(* Logix 5000 project; controller ChiaDynamix_PLC2 Emulate 5570 rev 30.12; software revision 30.00 *)

TASK T00_MainTask (continuous, watchdog 500 ms) : P00_MainProgram

MODULES
   Local : Emulate 5570 (ICP 5, rev 30.12)
      Entradas_Digitales : 1756-IB16 (ICP 3, rev 3.1, Input RPI 20 ms)
      Salidas_Digitales : vendor 1 type 7 code 16 (ICP 4, rev 3.1, Output RPI 20 ms)
      ChiaDynamix_PLC1 : Emulate 5570 (ICP 2, rev 30.1, $a5fb9b3a$ RPI 20 ms, $af09fea8$ RPI 20 ms)
      PLC_Seguridad : Emulate 5570 (ICP 6, rev 30.1, $68d98553$ RPI 20 ms)
END_MODULES

VAR_GLOBAL   (* controller tags *)
   Controles_Permisivos_Consumido : DINT;   // Señal de Seguridad que se recibe del PLC Seguridad
   COUNT : COUNTER[6] := ([0].PRE := 3, [0].ACC := 2, [1].PRE := 3, [1].ACC := 2);
        [1]   // Contador de Cajas Apiladas
        [0]   // Contador de Baldosas Apiladas
   Count_Baldosas_Producido : DINT; {produced}   // Señal que indica que el contador de baldosas ha sido alcanzado
   Count_Cajas_Producido : DINT; {produced}   // Señal que indica cuando el contador de cajas ha sido alcanzado
   FAB_CER_EME_002 : DINT; {produced}   // Botón de Emergencia del PLC2
   FAB_CER_HOMBRE_MUERTO_Producido : DINT; {produced}   // Dead Man Switch
   FAB_CER_RES_002 : DINT; {produced}   // Botón de Reset del PLC2
   FAB_CER_SCANNER_AREA_Producido : DINT; {produced}   // Scanner Area
   FAB_CER_STP_002 : DINT; {produced}   // Botón de Parada del PLC2
   FAB_CER_STR_002 : ALIAS FOR Local:3:I.Data.3;   // Botón de Start del PLC2
   FAB_CORTINAS_SEGURIDAD2_Producido : DINT; {produced}   // Cortinas de seguridad del PLC2
   FAB_INTERLOCK_PUERTA1_Producido : DINT; {produced}   // Interlock Puerta 1
   FAB_INTERLOCK_PUERTA2_Producido : DINT; {produced}   // Interlock Puerta 2
   MA_APILADO1 : ALIAS FOR Local:4:I.Data.6;   // Máquina Apiladora
   MA_EMPA : ALIAS FOR Local:4:I.Data.5;   // Máquina empacadora
   MA_QUAL : ALIAS FOR Local:4:I.Data.4;   // Máquina Qualitron
   MA_VINIPEL : ALIAS FOR Local:4:I.Data.3;   // Máquina Vinipel
   MOT_BAND_001 : ALIAS FOR Local:4:I.Data.2;   // Motor Banda transportadora
   MOT_BAND_DEF : ALIAS FOR Local:4:I.Data.1;   // Motor de banda transportadora de defectos
   MOT_BIFUR : ALIAS FOR Local:4:I.Data.0;   // Motor Palanca de Bifurcación
   POS_BAN_ROBOT2 : ALIAS FOR Local:3:I.Data.13;   // Sensor de posición ubicado en Robot
   POS_BAND_APILADOR : ALIAS FOR Local:3:I.Data.7;   // Sensor de posición ubicado en banda de la máquina apiladora
   POS_BAND_CAJA : ALIAS FOR Local:3:I.Data.6;   // Sensor de posición ubicado en banda del empacado de cajas
   POS_BAND_DEF : ALIAS FOR Local:3:I.Data.5;   // Sensor de posición ubicado en final de banda de defectuosos
   POS_BAND_QUAL : ALIAS FOR Local:3:I.Data.4;   // Sensor de posición ubicado en banda del proceso de Qualitron
   Q : BOOL[32] := ([10] := 1);
        [11]   // Memorias Virtual que activa Motor
        [14]   // Memorias Virtual que activa Motor
        [12]   // Memoria Virtual que activa palanca de bifurcación
        [15]   // Memoria Virtual que activa Máquina Empacadora
   Q10_Producido : DINT; {produced}   // Memoria virtual que activa Máquina Qualitrón
   Q13_Producido : DINT; {produced}   // Memoria Virtual activa Máquina Apiladora
   Q155 : BOOL;   // Memorias Virtual que activa Motor
   Q16_Producido : DINT; {produced}   // Memoria Virtual que activa Rutina del Robot
   Q17_Producido : DINT; {produced}   // Memoria virtual que activa máquina de Vinipel
   Q1_Consumido : DINT;   // Memoria Virtual Q1 que se recibe del PLC1
   Q9_Consumido : DINT;   // Memoria Virtual Q9 que se consume del PLC1
   ROUT_ROBOT2 : ALIAS FOR Local:4:I.Data.7;   // Rutina de Robot 2
   SIGNAL_APILADO1 : DINT; {produced}   // Señal que indica que rutina del Robot 1 ha sido finalizada
   SIGNAL_DEFECT : INT;   // 1: Baldosa NO tiene defecto 2: Baldosa SI tiene defecto
   SIGNAL_ECOPLAT : DINT; {produced}   // Señal que indica que el proceso de máquina de Vinipel ha finalizado
   SIGNAL_EMPA : BOOL;   // Señal que indica que el proceso de empacado finalizó
   SIGNAL_ROUT2 : DINT; {produced}   // Señal que indica que rutina del Robot 2 ha sido finalizada
   SIGNAL_STP : BOOL;   // Señal que indica que el botón de paro está activo
   TIMER : TIMER[6] := ([0].PRE := 30000, [1].PRE := 30000);
        [0]   // Timer de Proceso de Impresión
        [1]   // Timer de Proceso de Secado (Horno)
END_VAR

PROGRAM P00_MainProgram   (* main routine R00_MainRoutine *)

ROUTINE R00_MainRoutine   (* ladder *)
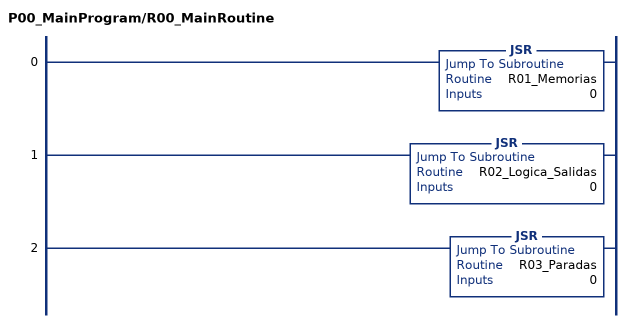
   0: JSR(R01_Memorias,0);
   1: JSR(R02_Logica_Salidas,0);
   2: JSR(R03_Paradas,0);
END_ROUTINE

ROUTINE R01_Memorias   (* ladder *)
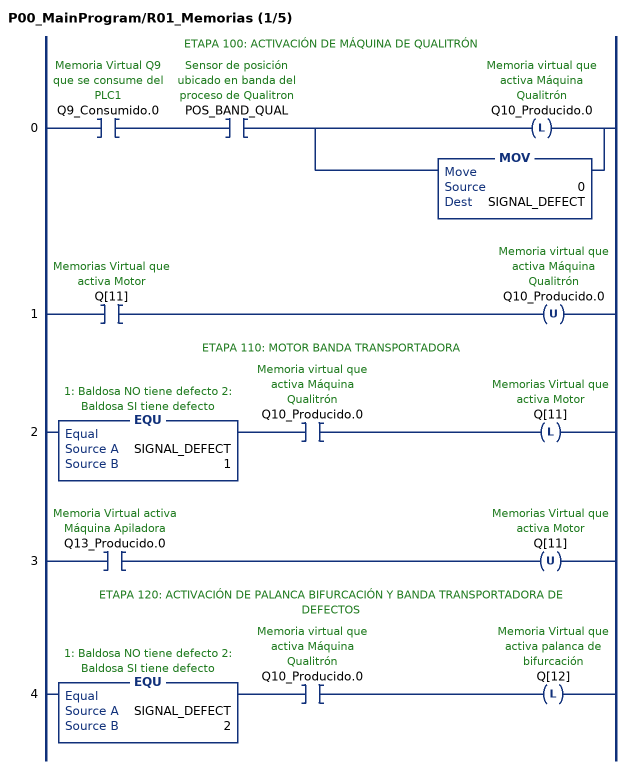
   // ETAPA 100: ACTIVACIÓN DE MÁQUINA DE QUALITRÓN
   0: XIC(Q9_Consumido.0)XIC(POS_BAND_QUAL)[OTL(Q10_Producido.0) ,MOV(0,SIGNAL_DEFECT) ];
   1: XIC(Q[11])OTU(Q10_Producido.0);
   // ETAPA 110: MOTOR BANDA TRANSPORTADORA
   2: EQU(SIGNAL_DEFECT,1)XIC(Q10_Producido.0)OTL(Q[11]);
   3: XIC(Q13_Producido.0)OTU(Q[11]);
   // ETAPA 120: ACTIVACIÓN DE PALANCA BIFURCACIÓN Y BANDA TRANSPORTADORA DE DEFECTOS
   4: EQU(SIGNAL_DEFECT,2)XIC(Q10_Producido.0)OTL(Q[12]);
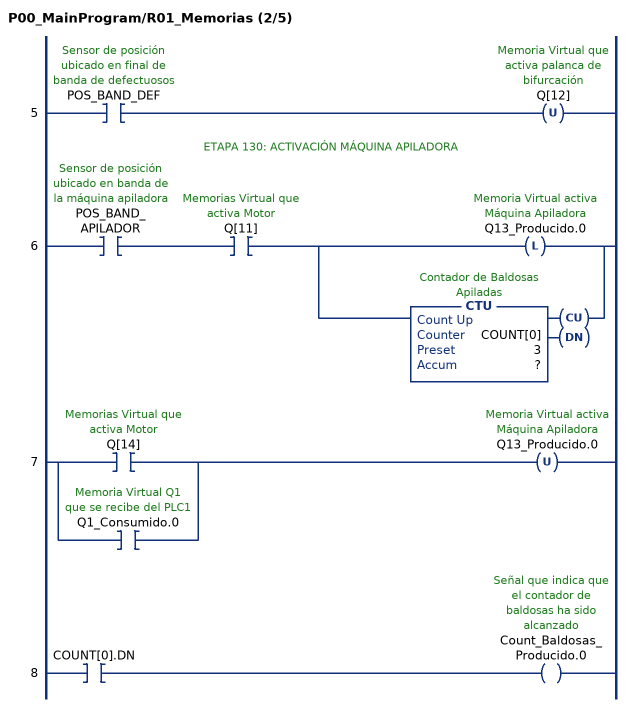
   5: XIC(POS_BAND_DEF)OTU(Q[12]);
   // ETAPA 130: ACTIVACIÓN MÁQUINA APILADORA
   6: XIC(POS_BAND_APILADOR)XIC(Q[11])[OTL(Q13_Producido.0) ,CTU(COUNT[0],?,?) ];
   7: [XIC(Q[14]) ,XIC(Q1_Consumido.0) ]OTU(Q13_Producido.0);
   8: XIC(COUNT[0].DN)OTE(Count_Baldosas_Producido.0);
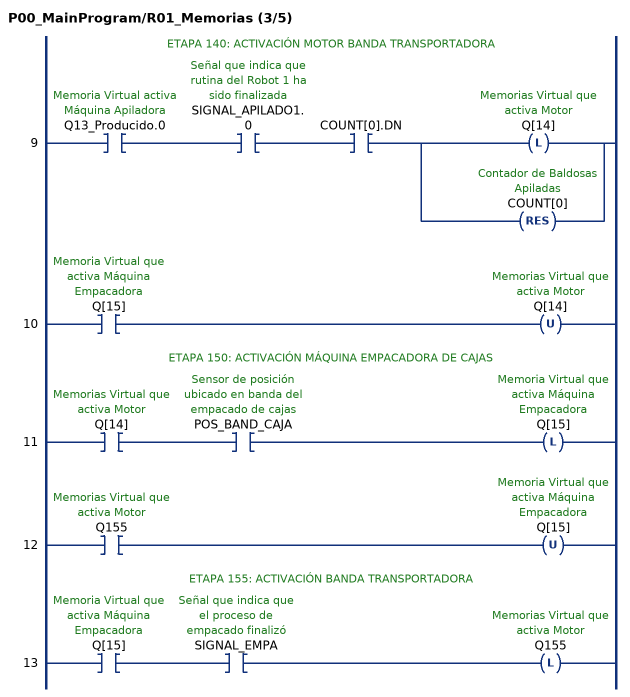
   // ETAPA 140: ACTIVACIÓN MOTOR BANDA TRANSPORTADORA
   9: XIC(Q13_Producido.0)XIC(SIGNAL_APILADO1.0)XIC(COUNT[0].DN)[OTL(Q[14]) ,RES(COUNT[0]) ];
   10: XIC(Q[15])OTU(Q[14]);
   // ETAPA 150: ACTIVACIÓN MÁQUINA EMPACADORA DE CAJAS
   11: XIC(Q[14])XIC(POS_BAND_CAJA)OTL(Q[15]);
   12: XIC(Q155)OTU(Q[15]);
   // ETAPA 155: ACTIVACIÓN BANDA TRANSPORTADORA
   13: XIC(Q[15])XIC(SIGNAL_EMPA)OTL(Q155);
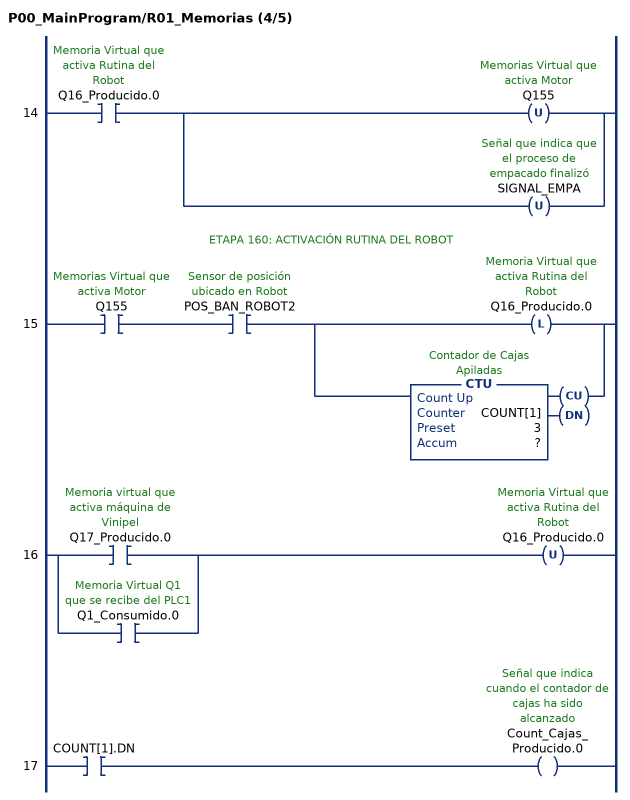
   14: XIC(Q16_Producido.0)[OTU(Q155) ,OTU(SIGNAL_EMPA) ];
   // ETAPA 160: ACTIVACIÓN RUTINA DEL ROBOT
   15: XIC(Q155)XIC(POS_BAN_ROBOT2)[OTL(Q16_Producido.0) ,CTU(COUNT[1],?,?) ];
   16: [XIC(Q17_Producido.0) ,XIC(Q1_Consumido.0) ]OTU(Q16_Producido.0);
   17: XIC(COUNT[1].DN)OTE(Count_Cajas_Producido.0);
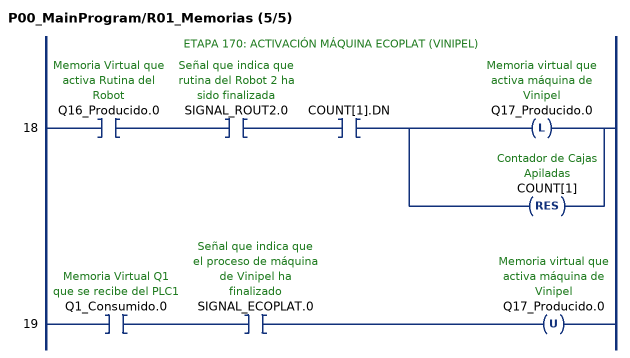
   // ETAPA 170: ACTIVACIÓN MÁQUINA ECOPLAT (VINIPEL)
   18: XIC(Q16_Producido.0)XIC(SIGNAL_ROUT2.0)XIC(COUNT[1].DN)[OTL(Q17_Producido.0) ,RES(COUNT[1]) ];
   19: XIC(Q1_Consumido.0)XIC(SIGNAL_ECOPLAT.0)OTU(Q17_Producido.0);
END_ROUTINE

ROUTINE R02_Logica_Salidas   (* ladder *)
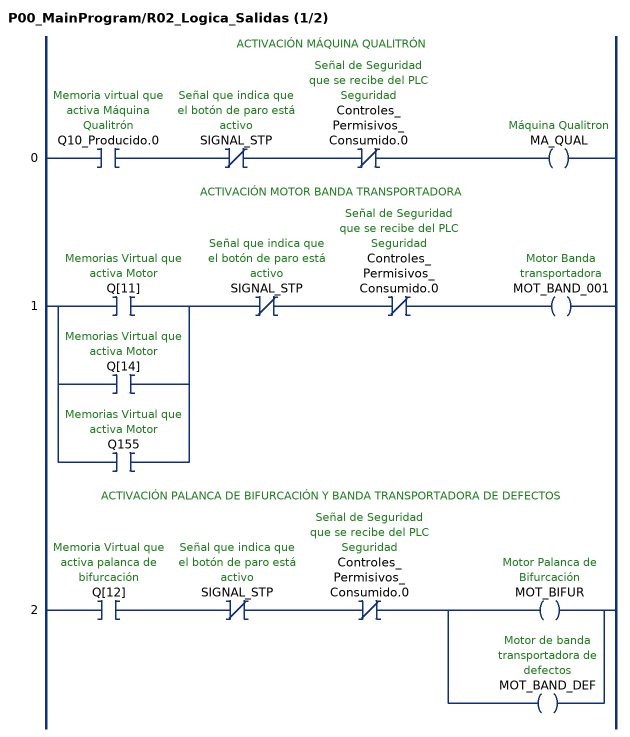
   // ACTIVACIÓN MÁQUINA QUALITRÓN
   0: XIC(Q10_Producido.0)XIO(SIGNAL_STP)XIO(Controles_Permisivos_Consumido.0)OTE(MA_QUAL);
   // ACTIVACIÓN MOTOR BANDA TRANSPORTADORA
   1: [XIC(Q[11]) ,XIC(Q[14]) ,XIC(Q155) ]XIO(SIGNAL_STP)XIO(Controles_Permisivos_Consumido.0)OTE(MOT_BAND_001);
   // ACTIVACIÓN PALANCA DE BIFURCACIÓN Y BANDA TRANSPORTADORA DE DEFECTOS
   2: XIC(Q[12])XIO(SIGNAL_STP)XIO(Controles_Permisivos_Consumido.0)[OTE(MOT_BIFUR) ,OTE(MOT_BAND_DEF) ];
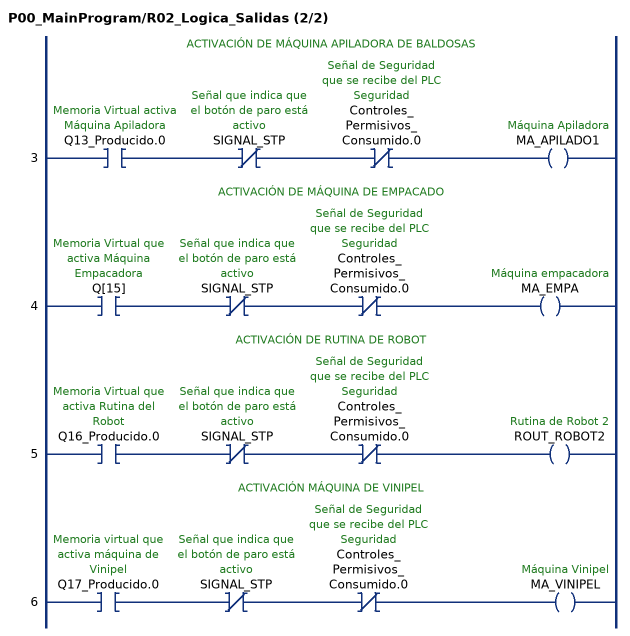
   // ACTIVACIÓN DE MÁQUINA APILADORA DE BALDOSAS
   3: XIC(Q13_Producido.0)XIO(SIGNAL_STP)XIO(Controles_Permisivos_Consumido.0)OTE(MA_APILADO1);
   // ACTIVACIÓN DE MÁQUINA DE EMPACADO
   4: XIC(Q[15])XIO(SIGNAL_STP)XIO(Controles_Permisivos_Consumido.0)OTE(MA_EMPA);
   // ACTIVACIÓN DE RUTINA DE ROBOT
   5: XIC(Q16_Producido.0)XIO(SIGNAL_STP)XIO(Controles_Permisivos_Consumido.0)OTE(ROUT_ROBOT2);
   // ACTIVACIÓN MÁQUINA DE VINIPEL
   6: XIC(Q17_Producido.0)XIO(SIGNAL_STP)XIO(Controles_Permisivos_Consumido.0)OTE(MA_VINIPEL);
END_ROUTINE

ROUTINE R03_Paradas   (* ladder *)
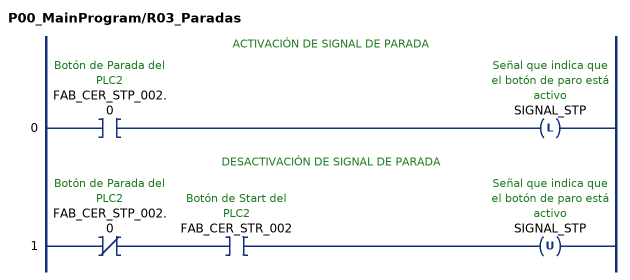
   // ACTIVACIÓN DE SIGNAL DE PARADA
   0: XIC(FAB_CER_STP_002.0)OTL(SIGNAL_STP);
   // DESACTIVACIÓN DE SIGNAL DE PARADA
   1: XIO(FAB_CER_STP_002.0)XIC(FAB_CER_STR_002)OTU(SIGNAL_STP);
END_ROUTINE
END_PROGRAM
